FUNCTION Celcius_Fahrenheit : REAL
VAR_INPUT
	fCelcius : REAL;
END_VAR
VAR
END_VAR

Celcius_Fahrenheit := fCelcius * 1.8 + 32.0;

END_FUNCTION

(* stored: Version 1.1.0.1, ProductVersion 3.1.4024.16
   POU Celcius_Fahrenheit: Id {7cd4b268-9c6e-4409-9255-3aac73334e94}, SpecialFunc None *)
